PROGRAM P_Task2
VAR
	fbTOF		: TOF;
	functest	:REAL;
	degval 		:REAL:=180;
END_VAR

fbTOF(
	IN		:=GVL_task2.stTimer2.bTimerStart2,
	PT		:=GVL_task2.stTimer2.tTimer2,
	Q		=>GVL_task2.stTimer2.bQStatus2,
	ET		=>GVL_task2.stTimer2.tElapsedTime2
);

GVL_task2.rMotor1Pos:=fDegToRad(rDegrees:=degval);

END_PROGRAM

(* stored: Version 1.1.0.1, ProductVersion 3.1.4024.12
   POU P_Task2: Id {b0fdee63-e475-4010-8043-331284731c8b}, SpecialFunc None *)
